FUNCTION_BLOCK FB_01
VAR_INPUT
END_VAR
VAR_OUTPUT
END_VAR
VAR
END_VAR

END_FUNCTION_BLOCK

(* stored: Version 1.1.0.1, ProductVersion 3.1.4024.12
   POU FB_01: Id {ddc71ac1-ee0a-4885-aaa7-7473e72484fa}, SpecialFunc None *)
